Omron CX-Programmer project NewProject (CX-Programmer 9.51)

# PLC My_first_project: CP1L L
; MyfirstProject

## Program NewProgram1 (cyclic task 0)
Local symbols
button_1 0.00 BOOL  ; comment
button_4 0.03 BOOL  ; comment
out_1 100.00 BOOL  ; out_1

### Section Section1

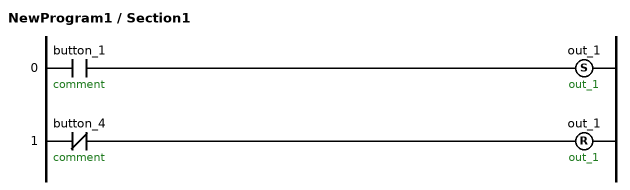
; rung 0
LD button_1  ; comment
SET out_1  ; out_1
; rung 1
LDNOT button_4  ; comment
RSET out_1  ; out_1

### Section END
; rung 0
END(001)